FUNCTION_BLOCK LfcPrint
  (* Standard: 61499-2 *)
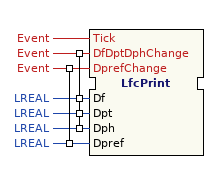
  EVENT_INPUT
    Tick;
    DfDptDphChange WITH Df, Dpt, Dph;
    DprefChange WITH Dpref;
  END_EVENT
  VAR_INPUT
    Df : LREAL;
    Dpt : LREAL;
    Dph : LREAL;
    Dpref : LREAL;
  END_VAR
END_FUNCTION_BLOCK
(* other elements stored in the file *)
(* Autogenerate Language=C ArbitraryText= #include <stdio.h> #include <stdlib.h> RunText= static int tickCount = 0; printf("%10f, %10f, %10f, %10f, %10f\r\n", tickCount * 0.0001, me->Dpref, me->Df, me->Dpt, me->Dph); tickCount++; *)
